TYPE ST_CraneKinematics :
STRUCT
END_STRUCT
END_TYPE

(* stored: Version 1.1.0.1, ProductVersion 3.1.4024.10
   DUT ST_CraneKinematics: Id {5295fcda-ae60-4776-a732-0e865c02fab3} *)
